// TIA Portal V20 export
TYPE "LER_typeCommunicationUnitStatus"
// stored: Access Published
   STRUCT
      specialFunctions : "LER_typeCommunicationSpecialFunctionsReelCut";
      mode : "LUC_typeModes";
      state : "LUC_typeStates";
      Alarms : "LAF_typeAlarms";
      commands : "LUC_typeStateCommands";
   END_STRUCT;
END_TYPE
